FUNCTION_BLOCK ASR_AX_SR_2 (* Event-driven bistable, bidirectional Socket (Set/Reset in, state back out via the same adapter) *)
  (* Standard: 61499-1 Annex A; Description: Copyright (c) 2026 HR Agrartechnik GmbH This program and the accompanying materials are made available under the terms of the Eclipse Public License 2.0 which is available at https://www.eclipse.org/legal/epl-2.0/ SPDX-License-Identifier: EPL-2.0 *)
  (* Version 1.0, 2026-09-03, Franz Höpfinger, HR Agrartechnik GmbH, wie ASR_AX_SR, aber mit bidirektionalem ASR_AX-Socket statt unidirektionalem ASR-Socket + separatem AX-Plug - der Zustand geht ueber denselben Adapter zurueck *)
  PACKAGE adapter::events::bidirectional;
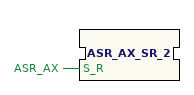
  SOCKETS
    S_R : adapter::types::bidirectional::ASR_AX; (* Set/Reset (in), Zustand (out) *)
  END_SOCKETS
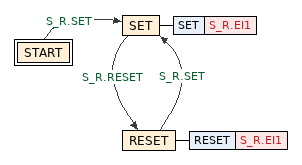
  EC_STATES
    START; (* Initial State *)
    SET : SET -> S_R.EI1;
    RESET : RESET -> S_R.EI1;
  END_STATES
  EC_TRANSITIONS
    START TO SET := S_R.SET;
    SET TO RESET := S_R.RESET;
    RESET TO SET := S_R.SET;
  END_TRANSITIONS
  ALGORITHM SET IN ST:
S_R.DI1 := TRUE;
  END_ALGORITHM
  ALGORITHM RESET IN ST:
S_R.DI1 := FALSE;
  END_ALGORITHM
END_FUNCTION_BLOCK
